//{attribute 'qualified_only'}
//{attribute 'strict'}
{attribute 'to_string'}

TYPE E_Util_Service_Req :
(
	Off			:= 0,
	On 			:= 1
//	Reset		:= 2
);
END_TYPE

(* stored: Version 1.1.0.1, ProductVersion 3.1.4024.12
   DUT E_Util_Service_Req: Id {d6dc575d-ec45-4850-9a51-cf2bd5d1ed73} *)
